PROGRAM ESC
VAR_INPUT
	
	sMotorspeed : STRING; // 'ESC1:value', 'ESC2:value'

END_VAR
VAR_OUTPUT
	
END_VAR
VAR
	fbescCommunication : FB_ESCcommunication;

	bESCerror : BOOL;
    ESCerrorID : ComError_t;
	
	currentcotrol : UINT :=0;
	previouscotrol : UINT :=0;
	timer: TON;
	
	
END_VAR

fbescCommunication(senddata := sMotorspeed, TxBuffer:=TxBufferEL6021, RxBuffer:=RxBufferEL6021,
bReceiveError => bESCerror, eReceiveErrorID =>ESCerrorID);

END_PROGRAM

(* stored: Version 1.1.0.1, ProductVersion 3.1.4024.13
   POU ESC: Id {ef45f950-70ba-4448-9518-507723000ff3}, SpecialFunc None *)
